(* IEC 61131-3 sources: std_i2980_v2.06_cp053/Source/IMM/ieccontrol/NozzleGeneral (part 5) *)

@F

@Trans @RT(7)Trans56 @F @T @F @F @T @F @TL(2)
TRUE

@RT(7)Trans56 @F
@Goto @RT(7)S_Ready @F @F

@Step @RT(6)Step45 @F @F @F @F @RT(0) @F
@AcbCont @RT(7)unnamed @F 0

@AltBranch @RT(3)alt @F 2
@TransSeq @RT(4)tseq @F 1
@Trans @RT(13)TNozzleNotFwd @F @T @F @F @T @F @TL(2)
NOT sv_bNozzleFwd

@RT(13)TNozzleNotFwd @F

@TransSeq @RT(4)tseq @F 4
@Trans @RT(12)TNozzleIsFwd @F @T @F @F @T @F @TL(2)
sv_bNozzleFwd

@RT(12)TNozzleIsFwd @F
@Step @RT(6)Step47 @F @F @F @F @RT(0) @F
@AcbCont @RT(7)unnamed @F 1
@Acb @RT(23)ASetContactPressBuildUp @F @T @RT(1)P @RT(0) @F @F @T @TL(2)
bContactPressBuildUp := TRUE;

@F

@Trans @RT(7)Trans71 @F @T @F @F @T @F @TL(2)
TRUE

@RT(7)Trans71 @F
@Goto @RT(24)S_CheckIfPressureBuildUp @F @F

@Step @RT(13)S_ProfileMove @F @F @F @F @RT(0) @F
@AcbCont @RT(7)unnamed @F 5
@Acb @RT(18)AResetProfileBlock @F @F @RT(1)P @RT(0) @F @F @F @F
@Acb @RT(15)AResetDetection @F @F @RT(1)P @RT(0) @F @F @F @F
@Acb @RT(11)aRunProfile @F @F @RT(1)N @RT(0) @F @F @F @F
@Acb @RT(18)ACheckContactPoint @F @F @RT(1)N @RT(0) @F @F @F @F
@Acb @RT(18)ACheckPointReached @F @F @RT(2)P0 @RT(0) @F @F @F @F

@Trans @RT(17)TProfileMoveReady @F @T @F @F @T @F @TL(2)
NOT abNozzleFwdProfile.aRun.bActive

@RT(17)TProfileMoveReady @F
@Step @RT(7)S_Check @F @F @F @F @RT(0) @F
@AcbCont @RT(7)unnamed @F 0

@AltBranch @RT(3)alt @F 2
@TransSeq @RT(4)tseq @F 1
@Trans @RT(15)TContactPointOk @F @T @F @F @T @F @TL(2)
bContactPointDetected

@RT(15)TContactPointOk @F

@TransSeq @RT(4)tseq @F 2
@Trans @RT(18)TContactPointNotOk @F @T @F @F @T @F @TL(2)
NOT bContactPointDetected

@RT(18)TContactPointNotOk @F
@Goto @RT(7)S_Ready @F @F

@Step @RT(14)S_NewPosOffset @F @F @F @F @RT(0) @F
@AcbCont @RT(7)unnamed @F 1
@Acb @RT(21)AActivateContactForce @F @T @RT(1)P @RT(0) @F @F @T @TL(2)
bContactPressBuildUp := TRUE;

@F

@Trans @RT(7)Trans45 @F @T @F @F @T @F @TL(2)
TRUE

@RT(7)Trans45 @F

@TransSeq @RT(4)tseq @F 11
@Trans @RT(12)TLimitSwitch @F @T @F @F @T @F @TL(2)
sv_MovementMode = nLimitSwitchDependent

@RT(12)TLimitSwitch @F
@Step @RT(18)S_CheckLimitSwitch @F @F @F @F @RT(0) @F
@AcbCont @RT(7)unnamed @F 1
@Acb @RT(8)Action21 @F @T @RT(1)N @RT(0) @F @F @T @TL(3)
dActiveTime := T#0s;
sv_NozzleFwdTimesAct.dActMoveTime := T#0s;

@F

@AltBranch @RT(3)alt @F 2
@TransSeq @RT(4)tseq @F 1
@Trans @RT(21)TLimitSwitchAvailable @F @T @F @F @T @F @TL(3)
mbLimitSwFwdLinked AND
NOT di_LimitSwitchFwd

@RT(21)TLimitSwitchAvailable @F

@TransSeq @RT(4)tseq @F 4
@Trans @RT(17)TStartSecondStage @F @T @F @F @T @F @TL(4)
mbLimitSwFwdLinked AND
di_LimitSwitchFwd

@RT(17)TStartSecondStage @F
@Step @RT(11)CheckLimits @F @F @F @F @RT(0) @F
@AcbCont @RT(7)unnamed @F 0

@AltBranch @RT(3)alt @F 3
@TransSeq @RT(4)tseq @F 1
@Trans @RT(12)TGoToTimeDep @F @T @F @F @T @F @TL(3)
NOT mbLimitSwFwd2Linked

@RT(12)TGoToTimeDep @F

@TransSeq @RT(4)tseq @F 2
@Trans @RT(18)TGoToSecLimitSwDep @F @T @F @F @T @F @TL(3)
mbLimitSwFwd2Linked AND
NOT di_LimitSwitchFwd2

@RT(18)TGoToSecLimitSwDep @F
@Goto @RT(16)S_ConstStage2Di2 @F @F

@TransSeq @RT(4)tseq @F 2
@Trans @RT(14)TNozzleInFront @F @T @F @F @T @F @TL(3)
mbLimitSwFwd2Linked
AND di_LimitSwitchFwd2

@RT(14)TNozzleInFront @F
@Goto @RT(29)S_ActivateContactFAfterLimSW2 @F @F

@Goto @RT(13)S_ConstStage2 @F @F

@Step @RT(13)S_ConstStage1 @F @F @F @F @RT(0) @F
@AcbCont @RT(7)unnamed @F 4
@Acb @RT(17)AResetConstStage1 @F @F @RT(1)P @RT(0) @F @F @F @F
@Acb @RT(17)ACheckVelCReached @F @F @RT(1)N @RT(0) @F @F @F @F
@Acb @RT(15)AS2PreOutputMax @F @F @RT(1)N @RT(0) @F @F @F @F
@Acb @RT(15)aRunConstStage1 @F @F @RT(1)N @RT(0) @F @F @F @F

@AltBranch @RT(3)alt @F 3
@TransSeq @RT(4)tseq @F 1
@Trans @RT(19)TLimitSwitchReached @F @T @F @F @T @F @TL(4)
di_LimitSwitchFwd AND
bVelC1Reached AND
NOT mbLimitSwFwd2Linked

@RT(19)TLimitSwitchReached @F

@TransSeq @RT(4)tseq @F 6
@Trans @RT(20)TGoToNextLimitSwitch @F @T @F @F @T @F @TL(4)
mbLimitSwFwd2Linked AND
di_LimitSwitchFwd AND
bVelC1Reached

@RT(20)TGoToNextLimitSwitch @F
@Step @RT(16)S_ConstStage2Di2 @F @F @T @F @RT(0) @F
@AcbCont @RT(7)unnamed @F 3
@Acb @RT(20)AResetConstStage2DI2 @F @F @RT(1)P @RT(0) @F @F @F @F
@Acb @RT(16)AStopConstStage1 @F @F @RT(1)N @RT(0) @F @F @F @F
@Acb @RT(18)aRunConstStage1To2 @F @F @RT(1)N @RT(0) @F @F @F @F

@Trans @RT(7)Trans44 @F @T @F @F @T @F @TL(3)
((NOT abNozzleFwdConstStage2.aRun.bActive)
AND(NOT abNozzleFwdConstStage1.aRun.bActive))

@RT(7)Trans44 @F
@Step @RT(29)S_ActivateContactFAfterLimSW2 @F @F @T @F @RT(0) @F
@AcbCont @RT(7)unnamed @F 1
@Acb @RT(24)AActivateConFAfterLimSW2 @F @T @RT(1)P @RT(0) @F @F @T @TL(4)
IF di_LimitSwitchFwd2 THEN
   bContactPressBuildUp := TRUE;
END_IF;

@F

@Trans @RT(7)Trans67 @F @T @F @F @T @F @TL(2)
TRUE

@RT(7)Trans67 @F
@Goto @RT(8)S_PreOut @F @F

@TransSeq @RT(4)tseq @F 2
@Trans @RT(7)Trans35 @F @T @F @F @T @T @TL(2)
NOT abNozzleFwdConstStage1.aRun.bActive

@RT(7)Trans35 @F
@Goto @RT(8)S_PreOut @F @F

@Step @RT(13)S_ConstStage2 @F @F @T @F @RT(0) @F
@AcbCont @RT(7)unnamed @F 3
@Acb @RT(17)AResetConstStage2 @F @F @RT(1)P @RT(0) @F @F @F @F
@Acb @RT(16)AStopConstStage1 @F @F @RT(1)N @RT(0) @F @F @F @F
@Acb @RT(15)aRunConstStage2 @F @F @RT(1)N @RT(0) @F @F @F @F

@Trans @RT(17)TConstStage2Ready @F @T @F @F @T @F @TL(3)
    (NOT abNozzleFwdConstStage2.aRun.bActive)
AND (NOT abNozzleFwdConstStage1.aRun.bActive)

@RT(17)TConstStage2Ready @F
@Step @RT(29)S_ActivateContactFAfterLimSW1 @F @F @F @F @RT(0) @F
@AcbCont @RT(7)unnamed @F 1
@Acb @RT(24)AActivateConFAfterLimSW1 @F @T @RT(1)P @RT(0) @F @F @T @TL(4)
IF (sv_dNozzleFwdStage2Act >= sv_dNozzleFwdStage2Set) THEN
   bContactPressBuildUp := TRUE;
END_IF;

@F

@Trans @RT(7)Trans68 @F @T @F @F @T @F @TL(2)
TRUE

@RT(7)Trans68 @F
@Step @RT(8)S_PreOut @F @F @T @F @RT(0) @F
@AcbCont @RT(7)unnamed @F 1
@Acb @RT(13)AS2PreOutput0 @F @F @RT(1)N @RT(0) @F @F @F @F

@Trans @RT(7)Trans21 @F @T @F @F @T @F @TL(2)
TRUE

@RT(7)Trans21 @F

@TransSeq @RT(4)tseq @F 5
@Trans @RT(9)TTimeMode @F @T @F @F @T @F @TL(2)
sv_MovementMode = nMoveTimeDependent

@RT(9)TTimeMode @F
@Step @RT(11)S_ConstTime @F @F @F @F @RT(0) @F
@AcbCont @RT(7)unnamed @F 3
@Acb @RT(6)AReset @F @F @RT(1)P @RT(0) @F @F @F @F
@Acb @RT(13)aRunConstTime @F @F @RT(1)N @RT(0) @F @F @F @F
@Acb @RT(18)ASetFwdTimeReached @F @F @RT(1)N @RT(0) @F @F @F @F

@Trans @RT(14)TTimeMoveReady @F @T @F @F @T @F @TL(2)
NOT abNozzleFwdConstStage2.aRun.bActive

@RT(14)TTimeMoveReady @F
@Step @RT(30)S_ActivateConFAfterTimeElapsed @F @F @F @F @RT(0) @F
@AcbCont @RT(7)unnamed @F 1
@Acb @RT(29)AActivateConFAfterTimeElapsed @F @T @RT(1)P @RT(0) @F @F @T @TL(2)
bContactPressBuildUp := sv_bFwdTimeReached;

@F

@Trans @RT(7)Trans64 @F @T @F @F @T @F @TL(2)
TRUE

@RT(7)Trans64 @F

@Step @RT(24)S_CheckIfPressureBuildUp @F @F @T @F @RT(0) @F
@AcbCont @RT(7)unnamed @F 0

@AltBranch @RT(3)alt @F 2
@TransSeq @RT(4)tseq @F 3
@Trans @RT(16)TMoveFwdContactF @F @T @F @F @T @F @TL(3)
g_MoveCtrl.pData^.MoveId = cMoveFwdContactF
AND bContactPressBuildUp

@RT(16)TMoveFwdContactF @F
@Step @RT(23)S_NozzlePressureBuildup @F @F @F @F @RT(0) @F
@AcbCont @RT(7)unnamed @F 2
@Acb @RT(23)AResetConstBuildUpPress @F @F @RT(1)P @RT(0) @F @F @F @F
@Acb @RT(21)aRunConstBuildUpPress @F @F @RT(1)N @RT(0) @F @F @F @F

@Trans @RT(18)TPressBuiltUpReady @F @T @F @F @T @F @TL(2)
NOT abNozzleFwdPressBuildUp.aRun.bActive

@RT(18)TPressBuiltUpReady @F

@TransSeq @RT(4)tseq @F 3
@Trans @RT(8)TMoveFwd @F @T @F @F @T @F @TL(3)
g_MoveCtrl.pData^.MoveId = cMoveFwd
OR NOT bContactPressBuildUp

@RT(8)TMoveFwd @F
@Step @RT(15)S_AdaptDuration @F @F @F @F @RT(0) @F
@AcbCont @RT(7)unnamed @F 1
@Acb @RT(18)ADurationReference @F @F @RT(1)P @RT(0) @F @F @F @F

@Trans @RT(7)Trans72 @F @T @F @F @T @F @TL(2)
TRUE

@RT(7)Trans72 @F

@Step @RT(7)S_Ready @F @F @T @F @RT(0) @F
@AcbCont @RT(7)unnamed @F 1
@Acb @RT(6)AReady @F @T @RT(1)P @RT(0) @F @F @T @TL(5)
bReady := TRUE;
fbSetMovementState(MoveId   := g_MoveCtrl.pData^.MoveId,
                   MoveDir  := g_MoveCtrl.pData^.MoveDir,
                   State    := nInactive);

@F

@Trans @RT(6)TReady @F @T @T @T @T @T @TL(2)
TRUE

@RT(6)TReady @F

@END_SfcData
@SaActions 33
@SaText @RT(16)AResetConstBlock 1 @TL(7)
(**************************************** WARNING ********************************************
 *** The KEBA Kemro K2 System including software is not intended for safety control tasks! ***
 ***                       For further information see Comment tab!                        ***
 *********************************************************************************************)

abNozzleFwdConstSetup.aRun(bStart := FALSE);

@SaText @RT(18)AResetProfileBlock 1 @TL(8)
(**************************************** WARNING ********************************************
 *** The KEBA Kemro K2 System including software is not intended for safety control tasks! ***
 ***                       For further information see Comment tab!                        ***
 *********************************************************************************************)

abNozzleFwdProfile.aRun(bStart := FALSE);

@SaText @RT(17)AResetConstStage1 1 @TL(8)
(**************************************** WARNING ********************************************
 *** The KEBA Kemro K2 System including software is not intended for safety control tasks! ***
 ***                       For further information see Comment tab!                        ***
 *********************************************************************************************)

abNozzleFwdConstStage1.aRun(bStart := FALSE);
bStage1Runned := TRUE;

@SaText @RT(17)AResetConstStage2 1 @TL(10)
(**************************************** WARNING ********************************************
 *** The KEBA Kemro K2 System including software is not intended for safety control tasks! ***
 ***                       For further information see Comment tab!                        ***
 *********************************************************************************************)
dActiveTime := sv_NozzleFwdTimesAct.dActMoveTime;
abNozzleFwdConstStage2.aRun(bStart := FALSE);

//set move time
abNozzleFwdConstStage2.aSetMoveTime(dSetMoveTime := sv_dNozzleFwdStage2Set);

@SaText @RT(16)AResetCalibBlock 1 @TL(14)
(**************************************** WARNING ********************************************
 *** The KEBA Kemro K2 System including software is not intended for safety control tasks! ***
 ***                       For further information see Comment tab!                        ***
 *********************************************************************************************)

bError := FALSE;
abNozzleFwdCalib.aRun(bStart := FALSE,
                      LintabPoint := sv_TmpLintabPoint);
IF abNozzleFwdCalib.aRun.bError THEN
   sv_CalibState.Status := tnCalibState_Error;
   bError := TRUE;
   dummy := Print("Calib Error: Reset calib block failed");
END_IF;

@SaText @RT(17)ACheckVelCReached 1 @TL(2)
bVelC1Reached := (ABS(sv_rVelocityAbs - sv_ConstFwdStage1.Velocity.Output.rOutputValue) < 0.1);

@SaText @RT(13)AS2PreOutput0 1 @TL(5)
bStage1Runned := FALSE;

sv_ConstFwdStage2.Pressure.PreOutput.rOutputValue := 0.0;
sv_ConstFwdStage2.Velocity.PreOutput.rOutputValue := 0.0;

@SaText @RT(15)AS2PreOutputMax 1 @TL(7)

IF bVelC1Reached THEN
  sv_ConstFwdStage2.Pressure.PreOutput.rOutputValue := sv_ConstFwdStage1.Pressure.Output.rOutputValue;
  sv_ConstFwdStage2.Velocity.PreOutput.rOutputValue := sv_ConstFwdStage1.Velocity.Output.rOutputValue;
END_IF;

@SaText @RT(16)AStopConstStage1 1 @TL(7)
(**************************************** WARNING ********************************************
 *** The KEBA Kemro K2 System including software is not intended for safety control tasks! ***
 ***                       For further information see Comment tab!                        ***
 *********************************************************************************************)

abNozzleFwdConstStage1.aRun(bStop:=TRUE);

@SaText @RT(16)ACheckCalibError 1 @TL(5)
IF bError THEN
   sv_CalibState.Status := tnCalibState_Error;
   dummy := Print("Calib Error: %i", iErrorInfo);
END_IF;

@SaText @RT(17)AResetAdjustBlock 1 @TL(14)
(**************************************** WARNING ********************************************
 *** The KEBA Kemro K2 System including software is not intended for safety control tasks! ***
 ***                       For further information see Comment tab!                        ***
 *********************************************************************************************)

//init supervision time
fbTSupervisionTime(IN := FALSE,
                   PT := sv_dMaxNozzleAdjustTime);

abNozzleFwdConstAdjust.aRun(bStart := FALSE);
bAutoAdjustAllowed := TRUE;

sv_rNozzlePositionOffset := 0.0;

@SaText @RT(16)AResetStandStill 1 @TL(6)
bStandStill := FALSE;

IF NOT mbLimitSwFwdLinked THEN
   fbStandStill(bDoCalib := FALSE);
END_IF;

@SaText @RT(17)ADetectStandStill 1 @TL(22)
(**************************************** WARNING ********************************************
 *** The KEBA Kemro K2 System including software is not intended for safety control tasks! ***
 ***                       For further information see Comment tab!                        ***
 *********************************************************************************************)

IF NOT bStandStill THEN
   IF mbLimitSwFwdLinked THEN
      bStandStill := di_LimitSwitchFwd;
   ELSE
      fbStandStill(rActVoltage := ai_Position,
                   bDoCalib := TRUE,
                   dCalibTime := sv_dSetStandstillDetectionTime,
                   rMaxVoltageDiff := sv_rMaxVoltageDiff,
                   bStandStill => bStandStill);
   END_IF;
END_IF;

@SaText @RT(16)ASetNozzleOffset 1 @TL(21)
(**************************************** WARNING ********************************************
 *** The KEBA Kemro K2 System including software is not intended for safety control tasks! ***
 ***                       For further information see Comment tab!                        ***
 *********************************************************************************************)

//calculate offset
//attention: offset is normally negative
sv_rNozzlePositionOffset := sv_rNozzlePositionOffset - sv_rNozzlePosition;

sv_rNozzleStrokePlaus := sv_rNozzleStroke + sv_rNozzlePositionOffset;

// automatically correct bwd profile if necessary
FOR i:=1 TO sv_NozzleBwdProfVis.Profile.iNoOfPoints + 1 DO
   sv_NozzleBwdProfVis.Profile.Points[i].rStartPos :=
         MIN(sv_NozzleBwdProfVis.Profile.Points[i].rStartPos, sv_rNozzleStrokePlaus);
END_FOR;

sv_bContactPointDetected := TRUE;
sv_bNozzleAdjHMI := FALSE;
SET_ALARM(erNozzleAdjustFinished);

@SaText @RT(23)AResetConstBuildUpPress 1 @TL(12)
(**************************************** WARNING ********************************************
*** The KEBA Kemro K2 System including software is not intended for safety control tasks! ***
***                       For further information see Comment tab!                        ***
*********************************************************************************************)

abNozzleFwdPressBuildUp.aRun(bStart := FALSE);

//set move time
abNozzleFwdPressBuildUp.aSetMoveTime(dSetMoveTime := sv_dNozzleFwdContactFSet);

sv_NozzleFwdContactFData.pdHoldDuration := @sv_dNozzleFwdContactFSet;

@SaText @RT(15)AResetDetection 1 @TL(11)
(**************************************** WARNING ********************************************
 *** The KEBA Kemro K2 System including software is not intended for safety control tasks! ***
 ***                       For further information see Comment tab!                        ***
 *********************************************************************************************)

bStandStill := FALSE;
fbStandStill(bDoCalib := FALSE);
fbRTrigStandstill(CLK := FALSE);
bContactPointDetected := FALSE;
bContactPointDetError := FALSE;

@SaText @RT(18)ACheckPointReached 1 @TL(18)
(**************************************** WARNING ********************************************
 *** The KEBA Kemro K2 System including software is not intended for safety control tasks! ***
 ***                       For further information see Comment tab!                        ***
 *********************************************************************************************)

IF abNozzleFwdProfile.aRun.bTimeOut OR abNozzleFwdProfile.aRun.bError THEN
   //timeout or error during profile movement
   bContactPointDetected := FALSE;
ELSIF (((sv_rNozzlePosition > sv_rPosOffsetTolerance) AND bStandStill)
   OR (sv_rNozzlePosition <= -sv_rPosOffsetTolerance)) THEN
   //standstill out of tolerance or movement finished out of tolerance
   bContactPointDetected := FALSE;
   SET_ALARM(erContactPointOutOfTolerance);
ELSE
   //movement finished inside the tolerance
   bContactPointDetected := TRUE;
END_IF;

@SaText @RT(18)ACheckContactPoint 1 @TL(11)
(**************************************** WARNING ********************************************
 *** The KEBA Kemro K2 System including software is not intended for safety control tasks! ***
 ***                       For further information see Comment tab!                        ***
 *********************************************************************************************)

fbStandStill(rActVoltage := ai_Position,
             bDoCalib := TRUE,
             dCalibTime := t#500ms,
             rMaxVoltageDiff := sv_rMaxVoltageDiff,
             bStandStill => bStandStill);

@SaText @RT(18)ADurationReference 1 @TL(7)
(**************************************** WARNING ********************************************
*** The KEBA Kemro K2 System including software is not intended for safety control tasks! ***
***                       For further information see Comment tab!                        ***
*********************************************************************************************)

sv_NozzleFwdContactFData.pdHoldDuration := EMPTY;

@SaText @RT(6)AReset 1 @TL(10)
(**************************************** WARNING ********************************************
 *** The KEBA Kemro K2 System including software is not intended for safety control tasks! ***
 ***                       For further information see Comment tab!                        ***
 *********************************************************************************************)

abNozzleFwdConstStage2.aRun(bStart := FALSE);

//set move time
abNozzleFwdConstStage2.aSetMoveTime(dSetMoveTime := sv_dNozzleFwdStage2Set);

@SaText @RT(18)ASetFwdTimeReached 1 @TL(7)
(**************************************** WARNING ********************************************
 *** The KEBA Kemro K2 System including software is not intended for safety control tasks! ***
 ***                       For further information see Comment tab!                        ***
 *********************************************************************************************)

sv_bFwdTimeReached := (sv_dNozzleFwdStage2Act >= sv_dNozzleFwdStage2Set)

@SaText @RT(20)AResetConstStage2DI2 1 @TL(8)
(**************************************** WARNING ********************************************
 *** The KEBA Kemro K2 System including software is not intended for safety control tasks! ***
 ***                       For further information see Comment tab!                        ***
 *********************************************************************************************)

dActiveTime := sv_NozzleFwdTimesAct.dActMoveTime;
abNozzleFwdConstStage2.aRun(bStart := FALSE);

@SaText @RT(16)AResetIdentBlock 1 @TL(3)
abNozzleFwdStep.aRun(bStart := FALSE);

@SaText @RT(16)ATransducerCalib 1 @TL(28)
(**************************************** WARNING ********************************************
 *** The KEBA Kemro K2 System including software is not intended for safety control tasks! ***
 ***                       For further information see Comment tab!                        ***
 *********************************************************************************************)

abNozzleFwdCalib.aRun(bStop := bStop OR sv_bTransducerError,
                      bStart := TRUE,
                      rActVoltage := ai_Position,
                      rMaxVoltageDiff := sv_rMaxVoltageDiff,
                      dStandStillDetectTime := sv_dStandStillDetectTime,
                      LintabPoint := sv_TmpLintabPoint,
                      rSetValue := 0.0,
                      dDelayTimeOn := sv_NozzleFwdTimesSet.dSetDelayTimePump,
                      dDelayTimeOff := sv_NozzleFwdTimesSet.dSetDelayTimeValve,
                      bActive => sv_bOutputActive,
                      rOutputPre => sv_rPressureAbs,
                      rOutputVel => sv_rVelocityAbs,
                      bPreOutputReached => sv_bPreOutputReady,
                      iErrorInfo => iErrorInfo);
sv_bDoTransducerCalib := NOT (abNozzleFwdCalib.aRun.bPointDetected);
bError := abNozzleFwdCalib.aRun.bError OR bError;

abLintabApplyPres.aCalc(rX := sv_rPressureAbs,
                        rY => sv_rPressure);

abLintabApplyVel.aCalc(rX := sv_rVelocityAbs,
                       rY => sv_rVelocity);

@SaText @RT(11)AStepOutput 1 @TL(30)
(**************************************** WARNING ********************************************
 *** The KEBA Kemro K2 System including software is not intended for safety control tasks! ***
 ***                       For further information see Comment tab!                        ***
 *********************************************************************************************)

abNozzleFwdStep.aRun(bUsePosDetect := sv_rIdentPosition <> 0.0,
                     rPositionDown := (sv_rNozzlePosition + sv_rIdentPosition) * 0.5,
                     rLowOutput := sv_rMaxSpeedFwd * 0.1,
                     bStart := TRUE,
                     bStop := bStop,
                     bDirection := FALSE,
                     rActPos := sv_rNozzlePosition,
                     rTargetPos := sv_rIdentPosition,
                     dDelayTimeOn := sv_NozzleFwdTimesSet.dSetDelayTimePump,
                     dDelayTimeOff := sv_dSetDelayTimeOffFwd,
                     rPositionUp := sv_rNozzlePosition,
                     rHighOutput := sv_ConstFwdSetup.Velocity.Output.rOutputValue,
                     dMaxMoveTime := sv_NozzleFwdTimesSet.dMaxMoveTime,
                     rStopRamp := sv_rIdentStopRamp,
                     bActive => sv_bOutputActive,
                     rOutputPre => sv_rPressureAbs,
                     rOutputVel => sv_rVelocityAbs,
                     bPreOutputReached => sv_bPreOutputReady);

abLintabApplyPres.aCalc(rX := sv_rPressureAbs,
                        rY => sv_rPressure);

abLintabApplyVel.aCalc(rX := sv_rVelocityAbs,
                       rY => sv_rVelocity);

@SaText @RT(11)aRunProfile 1 @TL(28)
(**************************************** WARNING ********************************************
 *** The KEBA Kemro K2 System including software is not intended for safety control tasks! ***
 ***                       For further information see Comment tab!                        ***
 *********************************************************************************************)

abNozzleFwdProfile.aRun(bStop := bStop OR sv_bTransducerError OR bStandStill,
                        bStart := TRUE,
                        rActPosition := sv_rNozzlePosition,
                        dMaxMoveTime := sv_NozzleFwdTimesSet.dMaxMoveTime,
                        dDelayTimeOn := sv_NozzleFwdTimesSet.dSetDelayTimePump,
                        dDelayTimeOff := sv_NozzleFwdTimesSet.dSetDelayTimeValve,
                        DeadTime := sv_dSetDelayTimeOffFwd,
                        rSmoothFactor := sv_rSmoothFactor,
                        bActive => sv_bOutputActive,
                        iActiveStage => sv_iActiveStage,
                        bPreOutputReached => sv_bPreOutputReady);

b := WRITE_SVREAL_DIRECT(sv_rPressureAbs, abNozzleFwdProfile.aRun.rPressureOutput);
b := WRITE_SVREAL_DIRECT(sv_rVelocityAbs, abNozzleFwdProfile.aRun.rVelocityOutput);
b := WRITE_SV_DIRECT(sv_NozzleFwdTimesAct.dActMoveTime, abNozzleFwdProfile.aRun.dActMoveTime);

abLintabApplyPres.aCalc(rX := sv_rPressureAbs);
b := WRITE_SVREAL_DIRECT(sv_rPressure, abLintabApplyPres.aCalc.rY);

abLintabApplyVel.aCalc(rX := sv_rVelocityAbs);
b := WRITE_SVREAL_DIRECT(sv_rVelocity, abLintabApplyVel.aCalc.rY);

@SaText @RT(13)aRunConstTime 1 @TL(26)
(**************************************** WARNING ********************************************
 *** The KEBA Kemro K2 System including software is not intended for safety control tasks! ***
 ***                       For further information see Comment tab!                        ***
 *********************************************************************************************)

abNozzleFwdConstStage2.aRun(bStart := TRUE,
                            bStop := bStop,
                            bUsePosDetect := FALSE,
                            dMaxTime := sv_NozzleFwdTimesSet.dMaxMoveTime,
                            dDelayTimeOn := sv_NozzleFwdTimesSet.dSetDelayTimePump,
                            dDelayTimeOff := sv_NozzleFwdTimesSet.dSetDelayTimeValve,
                            bActive => sv_bOutputActive,
                            bPreOutputReached => sv_bPreOutputReady);

b := WRITE_SVREAL_DIRECT(sv_rPressureAbs, abNozzleFwdConstStage2.aRun.rOutputPre);
b := WRITE_SVREAL_DIRECT(sv_rVelocityAbs, abNozzleFwdConstStage2.aRun.rOutputVel);
b := WRITE_SV_DIRECT(sv_NozzleFwdTimesAct.dActMoveTime, abNozzleFwdConstStage2.aRun.dActTime);
b := WRITE_SV_DIRECT(sv_dNozzleFwdStage2Act, sv_NozzleFwdTimesAct.dActMoveTime);

abLintabApplyPres.aCalc(rX := sv_rPressureAbs);
b := WRITE_SVREAL_DIRECT(sv_rPressure, abLintabApplyPres.aCalc.rY);

abLintabApplyVel.aCalc(rX := sv_rVelocityAbs);
b := WRITE_SVREAL_DIRECT(sv_rVelocity, abLintabApplyVel.aCalc.rY);

@SaText @RT(15)aRunConstStage2 1 @TL(43)
(**************************************** WARNING ********************************************
 *** The KEBA Kemro K2 System including software is not intended for safety control tasks! ***
 ***                       For further information see Comment tab!                        ***
 *********************************************************************************************)

IF (bStage1Runned) THEN
   dDelayTimeOn := T#0s;
   dDelayTimeOff := T#0s;
ELSE
   dDelayTimeOn := sv_NozzleFwdTimesSet.dSetDelayTimePump;
   dDelayTimeOff := sv_NozzleFwdTimesSet.dSetDelayTimeValve;
END_IF;

abNozzleFwdConstStage2.aRun(dMaxTime := sv_NozzleFwdTimesSet.dMaxMoveTime - dActiveTime,
                            bStart := TRUE,
                            bStop := bStop,
                            bUsePosDetect := FALSE,
                            dDelayTimeOn := dDelayTimeOn,
                            dDelayTimeOff := dDelayTimeOff,
                            rOutputPre => tmpPressureAbs,
                            rOutputVel => tmpVelocityAbs,
                            bActive => sv_bOutputActive,
                            bPreOutputReached => sv_bPreOutputReady);
dActMoveTime := abNozzleFwdConstStage2.aRun.dActTime + dActiveTime;
b := WRITE_SV_DIRECT(sv_NozzleFwdTimesAct.dActMoveTime, dActMoveTime);
b := WRITE_SV_DIRECT(sv_dNozzleFwdStage2Act, abNozzleFwdConstStage2.aRun.dActTime);

// sv_bPreOutput must be true for 2nd cycle, then outputvalue is valid
IF (sv_bPreOutputReady AND bPreOutputOld) THEN
   b := WRITE_SVREAL_DIRECT(sv_rPressureAbs, tmpPressureAbs);
   b := WRITE_SVREAL_DIRECT(sv_rVelocityAbs, tmpVelocityAbs);
END_IF;

bPreOutputOld := sv_bPreOutputReady;

abLintabApplyPres.aCalc(rX := sv_rPressureAbs);
b := WRITE_SVREAL_DIRECT(sv_rPressure, abLintabApplyPres.aCalc.rY);

abLintabApplyVel.aCalc(rX := sv_rVelocityAbs);
b := WRITE_SVREAL_DIRECT(sv_rVelocity, abLintabApplyVel.aCalc.rY);

@SaText @RT(18)aRunConstStage1To2 1 @TL(42)
(**************************************** WARNING ********************************************
 *** The KEBA Kemro K2 System including software is not intended for safety control tasks! ***
 ***                       For further information see Comment tab!                        ***
 *********************************************************************************************)

IF (bStage1Runned) THEN
   dDelayTimeOn := T#0s;
   dDelayTimeOff := T#0s;
ELSE
   dDelayTimeOn := sv_NozzleFwdTimesSet.dSetDelayTimePump;
   dDelayTimeOff := sv_NozzleFwdTimesSet.dSetDelayTimeValve;
END_IF;

abNozzleFwdConstStage2.aRun(bStop := bStop OR di_LimitSwitchFwd2,
                            dMaxTime := (sv_NozzleFwdTimesSet.dMaxMoveTime - dActiveTime),
                            bStart := TRUE,
                            bUsePosDetect := FALSE,
                            dDelayTimeOn := dDelayTimeOn,
                            dDelayTimeOff := dDelayTimeOff,
                            rOutputPre => tmpPressureAbs,
                            rOutputVel => tmpVelocityAbs,
                            bActive => sv_bOutputActive,
                            bPreOutputReached => sv_bPreOutputReady);
dActMoveTime := abNozzleFwdConstStage2.aRun.dActTime + dActiveTime;
b := WRITE_SV_DIRECT(sv_NozzleFwdTimesAct.dActMoveTime, dActMoveTime);

// sv_bPreOutput must be true for 2nd cycle, then outputvalue is valid
IF (sv_bPreOutputReady AND bPreOutputOld) THEN
   b := WRITE_SVREAL_DIRECT(sv_rPressureAbs, tmpPressureAbs);
   b := WRITE_SVREAL_DIRECT(sv_rVelocityAbs, tmpVelocityAbs);
END_IF;

bPreOutputOld := sv_bPreOutputReady;

abLintabApplyPres.aCalc(rX := sv_rPressureAbs);
b := WRITE_SVREAL_DIRECT(sv_rPressure, abLintabApplyPres.aCalc.rY);

abLintabApplyVel.aCalc(rX := sv_rVelocityAbs);
b := WRITE_SVREAL_DIRECT(sv_rVelocity, abLintabApplyVel.aCalc.rY);

@SaText @RT(15)aRunConstStage1 1 @TL(32)
(**************************************** WARNING ********************************************
 *** The KEBA Kemro K2 System including software is not intended for safety control tasks! ***
 ***                       For further information see Comment tab!                        ***
 *********************************************************************************************)

abNozzleFwdConstStage1.aRun(bStop := bStop OR (di_LimitSwitchFwd AND NOT bVelC1Reached),
                            bStart := TRUE,
                            bUsePosDetect := FALSE,
                            dMaxTime := sv_NozzleFwdTimesSet.dMaxMoveTime,
                            dDelayTimeOn := sv_NozzleFwdTimesSet.dSetDelayTimePump,
                            dDelayTimeOff := sv_NozzleFwdTimesSet.dSetDelayTimeValve,
                            rOutputPre => tmpPressureAbs,
                            rOutputVel => tmpVelocityAbs,
                            bActive => sv_bOutputActive,
                            bPreOutputReached => sv_bPreOutputReady);

b := WRITE_SV_DIRECT(sv_NozzleFwdTimesAct.dActMoveTime, abNozzleFwdConstStage1.aRun.dActTime);

// sv_bPreOutput must be true for 2nd cycle, then outputvalue is valid
IF (sv_bPreOutputReady AND bPreOutputOld) THEN
   b := WRITE_SVREAL_DIRECT(sv_rPressureAbs, tmpPressureAbs);
   b := WRITE_SVREAL_DIRECT(sv_rVelocityAbs, tmpVelocityAbs);
END_IF;

bPreOutputOld := sv_bPreOutputReady;

abLintabApplyPres.aCalc(rX := sv_rPressureAbs);
b := WRITE_SVREAL_DIRECT(sv_rPressure, abLintabApplyPres.aCalc.rY);

abLintabApplyVel.aCalc(rX := sv_rVelocityAbs);
b := WRITE_SVREAL_DIRECT(sv_rVelocity, abLintabApplyVel.aCalc.rY);

@SaText @RT(14)aRunConstSetup 1 @TL(22)
(**************************************** WARNING ********************************************
 *** The KEBA Kemro K2 System including software is not intended for safety control tasks! ***
 ***                       For further information see Comment tab!                        ***
 *********************************************************************************************)

abNozzleFwdConstSetup.aRun(bStart := TRUE,
                           bStop := bStop,
                           bUsePosDetect := FALSE,
                           dDelayTimeOn := sv_NozzleFwdTimesSet.dSetDelayTimePump,
                           dDelayTimeOff := sv_NozzleFwdTimesSet.dSetDelayTimeValve,
                           rOutputPre => sv_rPressureAbs,
                           rOutputVel => sv_rVelocityAbs,
                           bActive => sv_bOutputActive,
                           dActTime => sv_NozzleFwdTimesAct.dActMoveTime,
                           bPreOutputReached => sv_bPreOutputReady);

abLintabApplyPres.aCalc(rX := sv_rPressureAbs,
                        rY => sv_rPressure);

abLintabApplyVel.aCalc(rX := sv_rVelocityAbs,
                       rY => sv_rVelocity);

@SaText @RT(21)aRunConstBuildUpPress 1 @TL(27)
(**************************************** WARNING ********************************************
 *** The KEBA Kemro K2 System including software is not intended for safety control tasks! ***
 ***                       For further information see Comment tab!                        ***
 *********************************************************************************************)

abNozzleFwdPressBuildUp.aRun(bStart := TRUE,
                             bStop := bStop,
                             bUsePosDetect := FALSE,
                             dMaxTime := sv_NozzleFwdTimesSet.dMaxMoveTime,
                             dDelayTimeOn := sv_NozzleFwdTimesSet.dSetDelayTimePump,
                             dDelayTimeOff := sv_NozzleFwdTimesSet.dSetDelayTimeValve,
                             bActive => sv_bOutputActive,
                             bPreOutputReached => sv_bPreOutputReady);

sv_bPressBuildUpActive := sv_bOutputActive;
b := WRITE_SVREAL_DIRECT(sv_rPressureAbs, abNozzleFwdPressBuildUp.aRun.rOutputPre);
b := WRITE_SVREAL_DIRECT(sv_rVelocityAbs, abNozzleFwdPressBuildUp.aRun.rOutputVel);
b := WRITE_SV_DIRECT(sv_dActPressureBuildUpTime, abNozzleFwdPressBuildUp.aRun.dActTime);
b := WRITE_SV_DIRECT(sv_dNozzleFwdContactFAct, sv_dActPressureBuildUpTime);

abLintabApplyPres.aCalc(rX := sv_rPressureAbs);
b := WRITE_SVREAL_DIRECT(sv_rPressure, abLintabApplyPres.aCalc.rY);

abLintabApplyVel.aCalc(rX := sv_rVelocityAbs);
b := WRITE_SVREAL_DIRECT(sv_rVelocity, abLintabApplyVel.aCalc.rY);

@SaText @RT(20)aRunConstAdjustSetup 1 @TL(25)
(**************************************** WARNING ********************************************
 *** The KEBA Kemro K2 System including software is not intended for safety control tasks! ***
 ***                       For further information see Comment tab!                        ***
 *********************************************************************************************)

abNozzleFwdConstAdjust.aRun(bStop := bStop OR bStandStill OR sv_bTransducerError OR NOT bAutoAdjustAllowed,
                            bStart := TRUE,
                            bUsePosDetect := FALSE,
                            dMaxTime := sv_NozzleFwdTimesSet.dMaxMoveTime,
                            dDelayTimeOn := sv_NozzleFwdTimesSet.dSetDelayTimePump,
                            dDelayTimeOff := sv_NozzleFwdTimesSet.dSetDelayTimeValve,
                            rOutputPre => sv_rPressureAbs,
                            rOutputVel => sv_rVelocityAbs,
                            bActive => sv_bOutputActive,
                            dActTime => sv_NozzleFwdTimesAct.dActMoveTime,
                            bPreOutputReached => sv_bPreOutputReady);

abLintabApplyPres.aCalc(rX := sv_rPressureAbs,
                        rY => sv_rPressure);

abLintabApplyVel.aCalc(rX := sv_rVelocityAbs,
                       rY => sv_rVelocity);

@SaTrans 0
@SaExits 0
@END_SfcBody

@@@BEG_Comment@@@
@TL(0)

@@@END_Comment@@@

@BEG_Body
@TL(8)
(**************************************** WARNING ********************************************
 *** The KEBA Kemro K2 System including software is not intended for safety control tasks! ***
 ***                       For further information see Comment tab!                        ***
 *********************************************************************************************)

//copy stroke to start position of first profile point
sv_NozzleFwdProfVis.Profile.Points[1].rStartPos := sv_rNozzleStroke;

@END_Body

@@@BEG_Comment@@@
@TL(0)

@@@END_Comment@@@

@BEG_Body
@TL(15)
fuName := GET_MY_FU_NAME();
variableName := CONCAT(fuName,'.Fwd.rSetPressure bar');
swoState := KSWO_AddVariable( Task := TaskAnalog,
                              Name := variableName,
                              Variable := sv_rPressureAbs);
variableName := CONCAT(fuName,'.Fwd.rSetVelocity mm/s');
swoState := KSWO_AddVariable( Task := TaskAnalog,
                              Name := variableName,
                              Variable := sv_rVelocityAbs);
variableName := CONCAT(fuName,'.Fwd.bActive');
swoState := KSWO_AddVariable( Task := TaskAnalog,
                              Name := variableName,
                              Variable := sv_bOutputActive);
STOP_PROCESS_ALGORITHM();

@END_Body

@@@BEG_Comment@@@
@TL(0)

@@@END_Comment@@@

@BEG_Body
@TL(12)
(**************************************** WARNING ********************************************
 *** The KEBA Kemro K2 System including software is not intended for safety control tasks! ***
 ***                       For further information see Comment tab!                        ***
 *********************************************************************************************)

IF sv_MovementMode = nMoveTimeDependent THEN
   sv_NozzleFwdContactFData.pdInjectDuration := @sv_dNozzleFwdStage2Set;
ELSE
   sv_NozzleFwdContactFData.pdInjectDuration := @sv_dCalculatedDurationFwd;
END_IF;

@END_Body

@@@BEG_Comment@@@
@TL(0)

@@@END_Comment@@@

@BEG_Body
@TL(8)
(**************************************** WARNING ********************************************
 *** The KEBA Kemro K2 System including software is not intended for safety control tasks! ***
 ***                       For further information see Comment tab!                        ***
 *********************************************************************************************)

//update sv_rNozzleStrokePlaus (used for plaus on HMI)
sv_rNozzleStrokePlaus := sv_rNozzleStroke + sv_rNozzlePositionOffset;

@END_Body

@@@BEG_Comment@@@
@TL(0)

@@@END_Comment@@@

@BEG_Body
@TL(5)
FOR i:= 3 TO 20 DO
    sv_NozzleFwdProfVis.Profile.Points[i].rVelRamp := sv_NozzleFwdProfVis.Profile.Points[2].rVelRamp;
END_FOR;

@END_Body

@@@BEG_Comment@@@
@TL(0)

@@@END_Comment@@@

@BEG_Body
@TL(21)
(**************************************** WARNING ********************************************
 *** The KEBA Kemro K2 System including software is not intended for safety control tasks! ***
 ***                       For further information see Comment tab!                        ***
 *********************************************************************************************)

//deactive movement NozzleFwdContactF in HA and FA mode
//if nozzle is already forward and contact force build up time is 0.0 sec
IF (sv_OperationMode = nSetup) OR (sv_OperationMode = nManual) OR (sv_dNozzleFwdContactFSet > t#0.0s) THEN
   sv_MoveFwdContactF.pbActivated := @sv_bTRUE;
ELSE
   //HA or FA active and set set for contact forec build up = 0 sec.
   IF ((sv_MovementMode = nMoveTimeDependent) AND sv_bFwdTimeReached) OR
      ((sv_MovementMode <> nMoveTimeDependent) AND sv_bNozzleFwd) THEN
      // nozzle is already forward -> deactivate
      sv_MoveFwdContactF.pbActivated := @sv_bFALSE;
   ELSE
      // nozzle not forward -> activate
      sv_MoveFwdContactF.pbActivated := @sv_bTRUE;
   END_IF;
END_IF;

@END_Body

@@@BEG_Comment@@@
@TL(0)

@@@END_Comment@@@
@END_Body

@END_Contents

(* ---- ABMovementAdmin.pu ---- *)
IMPORT_OVER_LISTFILE
 STOP_PROCESS_ALGORITHM
, WRITE_SV_DIRECT
, cMoveFwd
, cMoveBwd
, cCompShutOffNozzle
, cSubOpNozzleTransducer
, cMoveFwdContactF
, ABMoveBwd
, ABMoveFwd
, tsMoveCtrl
, ABOutputRequest
, tOptionId
, tnOperationMode
, tsCalibMovement
, tsRequiredPumps
, tsHydrMaxValues
, KAPPL_LintabData
, tsCylinderData
, ABCalcHydrMaxValues
, ABUpdateRelLintabPre
, ABUpdateRelLintabVel

END_IMPORT

ALGORITHM_BLOCK ABMovementAdmin #DUMMY_EDIT_BLOCK

SYSTEM_VAR
 sv_bInitStart : BOOL;
 sv_bDeviceStart : BOOL (* Start Device *);
 ai_Position : REAL;
 sv_Options : tOptionId;
 sv_bTransducerAvailable : BOOL;
 sv_iActiveStage : DINT;
 sv_iActiveStageFwd : DINT (* active profile stage mold close (fwd) *);
 sv_iActiveStageBwd : DINT (* active profile stage mold open (bwd) *);
 sv_bDeviceReady : BOOL;
 sv_OperationMode : tnOperationMode;
 sv_CalibState : tsCalibMovement;
 sv_dActFwdTime : TIME (* actual nozzle fwd time (includes contact force build up) *);
 sv_RequiredPumpsFwd : tsRequiredPumps;
 sv_RequiredPumpsBwd : tsRequiredPumps;
 sv_HydrMaxValuesFwd : tsHydrMaxValues (* hydraulic max values for nozzle fwd *);
 sv_HydrMaxValuesBwd : tsHydrMaxValues (* hydraulic max values for nozzle bwd *);
 sv_bInitDone : BOOL;
 sv_LintabOutFwdP : KAPPL_LintabData;
 sv_LintabOutFwdV : KAPPL_LintabData;
 sv_LintabOutBwdP : KAPPL_LintabData;
 sv_LintabOutBwdV : KAPPL_LintabData;
 sv_rMaxSpeedFwd : REAL;
 sv_rMaxSpeedBwd : REAL;
 sv_CylinderData : tsCylinderData;
 sv_rMaxPressureFwd : REAL;
 sv_rMaxPressureBwd : REAL;
 sv_rMaxSpeedFwdCalc : REAL;
 sv_rMaxSpeedBwdCalc : REAL;
 sv_rMaxSpeedFwdCalib : REAL;
 sv_rMaxSpeedBwdCalib : REAL;
 sv_rMaxSpeedReducePercent : REAL;
 sv_bFALSE : BOOL;
END_VAR

SYSTEM_OBJECT
 PU_Task_7 : TASK;
 TaskAnalog : TASK;
 EV_Task_1 : TASK;
 PU_Task_3 : TASK;
END_OBJECT

VAR_EXTERNAL
 g_MoveCtrl : tsMoveCtrl;
END_VAR

VAR
 abMoveBwd : ABMoveBwd;
 abMoveFwd : ABMoveFwd;
 abOutputRequest : ABOutputRequest;
 miDigitsToFloor : SINT := 2;
END_VAR

(*
Calls the registration-algo of every movementblock after the deviceregistration succeeded(sv_bInitStart->true)

*)

POSTUPDATE_ALGORITHM pInitStart ON PU_Task_7 WITH sv_bInitStart

VAR
 abCalcMaxValuesFwd : ABCalcHydrMaxValues;
 abCalcMaxValuesBwd : ABCalcHydrMaxValues;
END_VAR
#BEGIN_EDIT_BLOCK
(**************************************** WARNING ********************************************
 *** The KEBA Kemro K2 System including software is not intended for safety control tasks! ***
 ***                       For further information see Comment tab!                        ***
 *********************************************************************************************)

IF sv_bInitStart THEN

   //check if transducer is available
   sv_bTransducerAvailable := IS_LINKED(ai_Position);
   IF (sv_bTransducerAvailable) THEN
      sv_Options := sv_Options OR cSubOpNozzleTransducer;
      //set auto-calib transducer
      sv_CalibState.prInputSensor := @ai_Position;
   END_IF;

   //register and init nozzle bwd movement
   abMoveBwd.aRegister();
   abMoveBwd.aInit();

   //register and init nozzle fwd movement
   abMoveFwd.aRegister();
   abMoveFwd.aInit();

   //init calculation of hydraulic max values for nozzle fwd
   abCalcMaxValuesFwd.aInit(pRequiredPumps := @sv_RequiredPumpsFwd,
                            pHydrMaxValues := @sv_HydrMaxValuesFwd);

   //init calculation of hydraulic max values for nozzle bwd
   abCalcMaxValuesBwd.aInit(pRequiredPumps := @sv_RequiredPumpsBwd,
                            pHydrMaxValues := @sv_HydrMaxValuesBwd);

END_IF;

;#END_EDIT_BLOCK END_ALGORITHM

(*
Starts the algo paRun when sv_bDeviceStart is set by ABControl.
*)

POSTUPDATE_ALGORITHM pDeviceStart ON EV_Task_1 WITH sv_bDeviceStart

#BEGIN_EDIT_BLOCK
(**************************************** WARNING ********************************************
 *** The KEBA Kemro K2 System including software is not intended for safety control tasks! ***
 ***                       For further information see Comment tab!                        ***
 *********************************************************************************************)

IF sv_bDeviceStart THEN
   //start device
   START_PROCESS_ALGORITHM(paRun);
END_IF;

;#END_EDIT_BLOCK END_ALGORITHM

POSTUPDATE_ALGORITHM pInitRelLintabUpdater ON PU_Task_7 WITH sv_bInitDone

VAR
 abUpdateRelLintabPreFwd : ABUpdateRelLintabPre;
 abUpdateRelLintabVelFwd : ABUpdateRelLintabVel;
 abUpdateRelLintabPreBwd : ABUpdateRelLintabPre;
 abUpdateRelLintabVelBwd : ABUpdateRelLintabVel;
END_VAR
#BEGIN_EDIT_BLOCK
(**************************************** WARNING ********************************************
 *** The KEBA Kemro K2 System including software is not intended for safety control tasks! ***
 ***                       For further information see Comment tab!                        ***
 *********************************************************************************************)

abUpdateRelLintabPreFwd.aInit(pLintabOut := @sv_LintabOutFwdP,
                              prMaxPressure := @sv_rMaxPressureFwd,
                              prMaxHydrPressure := @sv_HydrMaxValuesFwd.rMaxPressure,
                              bUseForce := TRUE,
                              bFwd := TRUE,
                              pCylinderData := @sv_CylinderData);

abUpdateRelLintabVelFwd.aInit(pLintabOut := @sv_LintabOutFwdV,
                              prMaxSpeed := @sv_rMaxSpeedFwd,
                              prMaxSpeedCalc := @sv_rMaxSpeedFwdCalc,
                              prMaxSpeedCalib := @sv_rMaxSpeedFwdCalib,
                              prMaxSpeedReducePercent := @sv_rMaxSpeedReducePercent,
                              iMaxSpeedDigitsToFloor := miDigitsToFloor,
                              prAbsFlow := @sv_HydrMaxValuesFwd.rAbsFlow,
                              bFwd := TRUE,
                              pCylinderData := @sv_CylinderData);

abUpdateRelLintabPreBwd.aInit(pLintabOut := @sv_LintabOutBwdP,
                              prMaxPressure := @sv_rMaxPressureBwd,
                              prMaxHydrPressure := @sv_HydrMaxValuesBwd.rMaxPressure,
                              bUseForce := TRUE,
                              bFwd := FALSE,
                              pCylinderData := @sv_CylinderData);

abUpdateRelLintabVelBwd.aInit(pLintabOut := @sv_LintabOutBwdV,
                              prMaxSpeed := @sv_rMaxSpeedBwd,
                              prMaxSpeedCalc := @sv_rMaxSpeedBwdCalc,
                              prMaxSpeedCalib := @sv_rMaxSpeedBwdCalib,
                              prMaxSpeedReducePercent := @sv_rMaxSpeedReducePercent,
                              iMaxSpeedDigitsToFloor := miDigitsToFloor,
                              prAbsFlow := @sv_HydrMaxValuesBwd.rAbsFlow,
                              bFwd := FALSE,
                              pCylinderData := @sv_CylinderData);

;#END_EDIT_BLOCK END_ALGORITHM

(*
Calls depending on the MoveId and MoveDir the movementblock. g_MoveCtrl.MoveId/MoveDir are set by the Block ABControl after
evStart was received. The movement-block has to be called until the it returns abMoveXxx.aRun.bReady.
In case of hydraulic movements the output-request has to be done before starting the movement.
*)

PROCESS_ALGORITHM paRun ON TaskAnalog(5000)

VAR_TEMP
 dActFwdTime : TIME;
 b : BOOL;
END_VAR

(* IecGraph-Code *)

(* init step *)
INITIAL_STEP START:
Action18 (P);
END_STEP

ACTION Action18: #BEGIN_EDIT_BLOCK
b := WRITE_SV_DIRECT(sv_bDeviceStart, sv_bFALSE);

;#END_EDIT_BLOCK END_ACTION (*Action18*)

(* steps *)
STEP OUTPUT_REQUEST:
AOutputRequest (P);
ACheckOutput (N);
END_STEP

ACTION AOutputRequest: #BEGIN_EDIT_BLOCK
abOutputRequest.aRequest(pMoveData := g_MoveCtrl.pData,
                         AnaOutputMode := nAnaOutputModeMid);

;#END_EDIT_BLOCK END_ACTION (*AOutputRequest*)
ACTION ACheckOutput: #BEGIN_EDIT_BLOCK
abOutputRequest.aCheck();

;#END_EDIT_BLOCK END_ACTION (*ACheckOutput*)
STEP OUTPUT:
END_STEP

STEP BWD:
aBwd (N);
END_STEP

STEP FWD:
aFwd (N);
END_STEP

STEP READY:
Action2 (P);
END_STEP

ACTION Action2: #BEGIN_EDIT_BLOCK
abOutputRequest.aRelease(pMoveData := g_MoveCtrl.pData);
g_MoveCtrl.bReady := TRUE;
IF NOT sv_bDeviceStart THEN
    STOP_PROCESS_ALGORITHM();
END_IF;

;#END_EDIT_BLOCK END_ACTION (*Action2*)

(* transitions *)
GO_ON_TRANSITION TStart (* Trans12 *) FROM START TO OUTPUT_REQUEST :=  #BEGIN_EDIT_BLOCK
TRUE
;#END_EDIT_BLOCK
END_TRANSITION

TRANSITION Trans13 (* Trans13 *) FROM OUTPUT_REQUEST TO READY :=  #BEGIN_EDIT_BLOCK
g_MoveCtrl.bStop
;#END_EDIT_BLOCK
END_TRANSITION

GO_ON_TRANSITION Trans15 (* Trans15 *) FROM OUTPUT_REQUEST TO OUTPUT :=  #BEGIN_EDIT_BLOCK
abOutputRequest.aCheck.bReady
;#END_EDIT_BLOCK
END_TRANSITION

GO_ON_TRANSITION Trans9 (* Trans9 *) FROM OUTPUT TO BWD :=  #BEGIN_EDIT_BLOCK
g_MoveCtrl.pData^.MoveDir = cMoveBwd
;#END_EDIT_BLOCK
END_TRANSITION

GO_ON_TRANSITION TBwdReady (* Trans1 *) FROM BWD TO READY :=  #BEGIN_EDIT_BLOCK
abMoveBwd.aRun.bReady;
;#END_EDIT_BLOCK
END_TRANSITION

GO_ON_TRANSITION Trans2 (* Trans2 *) FROM OUTPUT TO FWD :=  #BEGIN_EDIT_BLOCK
g_MoveCtrl.pData^.MoveDir = cMoveFwd
;#END_EDIT_BLOCK
END_TRANSITION

GO_ON_TRANSITION TFwdReady (* Trans11 *) FROM FWD TO READY :=  #BEGIN_EDIT_BLOCK
abMoveFwd.aRun.bReady
;#END_EDIT_BLOCK
END_TRANSITION

TRANSITION Trans8 (* Trans8 *) FROM READY TO START :=  #BEGIN_EDIT_BLOCK
TRUE
;#END_EDIT_BLOCK
END_TRANSITION

(* end IecGraph-Code *)
(* sfc-code *)

(* stand alone actions *)
ACTION aBwd: #BEGIN_EDIT_BLOCK
(**************************************** WARNING ********************************************
 *** The KEBA Kemro K2 System including software is not intended for safety control tasks! ***
 ***                       For further information see Comment tab!                        ***
 *********************************************************************************************)

abMoveBwd.aRun(bStop := g_MoveCtrl.bStop);

;#END_EDIT_BLOCK END_ACTION (*aBwd*)
ACTION aFwd: #BEGIN_EDIT_BLOCK
abMoveFwd.aRun(bStop := g_MoveCtrl.bStop);

IF g_MoveCtrl.pData^.MoveId = cMoveFwdContactF THEN
   dActFwdTime := FWD.T;
   b := WRITE_SV_DIRECT(sv_dActFwdTime, dActFwdTime);
END_IF;

;#END_EDIT_BLOCK END_ACTION (*aFwd*)
(* end sfc-code *)

END_ALGORITHM

POSTUPDATE_ALGORITHM pActiveProfileStage ON PU_Task_3 WITH sv_iActiveStage,sv_bDeviceReady

#BEGIN_EDIT_BLOCK
(**************************************** WARNING ********************************************
 *** The KEBA Kemro K2 System including software is not intended for safety control tasks! ***
 ***                       For further information see Comment tab!                        ***
 *********************************************************************************************)

IF NOT sv_bDeviceReady THEN

   IF sv_OperationMode = nSetup THEN
      //movement in setup mode active
      //-> reset active stage information
      sv_iActiveStageFwd := 0;
      sv_iActiveStageBwd := 0;
   ELSE

      //nozzle movement in manual - half - or fullauto mode
      IF g_MoveCtrl.pData^.MoveDir = cMoveFwd THEN

         //reset bwd stage info if fwd movement is started
         sv_iActiveStageBwd := 0;

         IF sv_iActiveStage > 0 THEN
            sv_iActiveStageFwd := sv_iActiveStage;
         END_IF;

      ELSIF g_MoveCtrl.pData^.MoveDir = cMoveBwd THEN

         //reset Fwd stage info if bwd movement is started
         sv_iActiveStageFwd := 0;

         IF sv_iActiveStage > 0 THEN
            sv_iActiveStageBwd := sv_iActiveStage;
         END_IF;
      END_IF;
   END_IF;

END_IF;

;#END_EDIT_BLOCK END_ALGORITHM

END_ALGORITHM_BLOCK

#END_OF_IEC_PART

@Puma @IecEditor 6 97 @Pou 25
@@@BEG_Comment@@@

@@@END_Comment@@@

@BEG_Contents

@BEG_Func
@RT(17)FuncTreeContainer
2
@Var @RT(22)STOP_PROCESS_ALGORITHM @RT(0) @T @T @DERIVED 0 @F @RT(23)KEBA_STANDARD_PROCEDURE @F
@T
@BEG_Attrib
0 @RT(0) @RT(0)
@END_Attrib
1 1 @F @F @F @F

@Var @RT(15)WRITE_SV_DIRECT @RT(0) @T @T @DERIVED 0 @F @RT(22)KEBA_STANDARD_FUNCTION @F
@T
@BEG_Attrib
0 @RT(0) @RT(0)
@END_Attrib
1 1 @F @F @F @F

@END_Func

@BEG_Const
@RT(18)ConstTreeContainer
5
@Var @RT(8)cMoveFwd @RT(0) @T @F @DT @RT(4)DINT @RT(0) @T @T @BASIC 0 @F
@F @F
@T
@BEG_Attrib
0 @RT(2)12 @RT(16)movement forward
@END_Attrib
1 1 @F @F @F @F

@Var @RT(8)cMoveBwd @RT(0) @T @F @DT @RT(4)DINT @RT(0) @T @T @BASIC 0 @F
@F @F
@T
@BEG_Attrib
0 @RT(2)11 @RT(17)movement backward
@END_Attrib
1 1 @F @F @F @F

@Var @RT(18)cCompShutOffNozzle @RT(0) @T @F @DT @RT(4)DINT @RT(0) @T @T @BASIC 0 @F
@F @F
@T
@BEG_Attrib
0 @RT(3)138 @RT(28)Component Shutter for Nozzle
@END_Attrib
1 1 @F @F @F @F

@Var @RT(22)cSubOpNozzleTransducer @RT(0) @T @F @DT @RT(5)DWORD @RT(0) @T @T @BASIC 0 @F
@F @F
@T
@BEG_Attrib
0 @RT(6)16#100 @RT(21)Nozzle has transducer
@END_Attrib
1 1 @F @F @F @F

@Var @RT(16)cMoveFwdContactF @RT(0) @T @F @DT @RT(4)DINT @RT(0) @T @T @BASIC 0 @F
@F @F
@T
@BEG_Attrib
0 @RT(2)66 @RT(45)nozzle forward with building up contact force
@END_Attrib
1 1 @F @F @F @F

@END_Const

@BEG_Export

@BEG_Kind
@ALGORITHM_BLOCK @RT(15)ABMovementAdmin @STRUCTURED_TEXT
@RT(0) @RT(0) @RT(0)
@END_Kind

@BEG_Dcl
@RT(16)DclTreeContainer
41
@Var @RT(9)abMoveBwd @RT(0) @T @T @DERIVED 0 @T @T @DT @RT(9)ABMoveBwd @RT(0) @T @T @UNKNOWN 0 @F
@F @F
@T
@BEG_Attrib
3 @RT(0) @RT(0) @RT(0)
@END_Attrib
1 0 @F @F @F @F

@Var @RT(9)abMoveFwd @RT(0) @T @T @DERIVED 0 @T @T @DT @RT(9)ABMoveFwd @RT(0) @T @T @UNKNOWN 0 @F
@F @F
@T
@BEG_Attrib
3 @RT(0) @RT(0) @RT(0)
@END_Attrib
1 0 @F @F @F @F

@Var @RT(13)sv_bInitStart @RT(0) @T @F @DT @RT(4)BOOL @RT(0) @T @T @BASIC 0 @F
@F @F
@T
@BEG_Attrib
3 @RT(0) @RT(0) @RT(0)
@END_Attrib
1 8 @F @F @F @F

@Var @RT(15)sv_bDeviceStart @RT(0) @T @F @DT @RT(4)BOOL @RT(0) @T @T @BASIC 0 @F
@F @F
@T
@BEG_Attrib
3 @RT(0) @RT(12)Start Device @RT(0)
@END_Attrib
1 8 @F @F @F @F

@Var @RT(10)g_MoveCtrl @RT(0) @T @T @DERIVED 0 @T @T @DT @RT(10)tsMoveCtrl @RT(0) @T @T @UNKNOWN 0 @F
@F @F
@T
@BEG_Attrib
3 @RT(0) @RT(0) @RT(0)
@END_Attrib
1 6 @F @F @F @F

@Var @RT(9)PU_Task_7 @RT(0) @T @T @RENAMED 0 @T @T @DT @RT(4)TASK @RT(0) @T @T @BASIC 0 @F
@F @F
@T
@BEG_Attrib
3 @RT(0) @RT(0) @RT(0)
@END_Attrib
1 7 @F @F @F @F

@Var @RT(15)abOutputRequest @RT(0) @T @T @DERIVED 0 @T @T @DT @RT(15)ABOutputRequest @RT(0) @T @T @UNKNOWN 0 @F
@F @F
@T
@BEG_Attrib
3 @RT(0) @RT(0) @RT(0)
@END_Attrib
1 0 @F @F @F @F

@Var @RT(10)TaskAnalog @RT(0) @T @T @RENAMED 0 @T @T @DT @RT(4)TASK @RT(0) @T @T @BASIC 0 @F
@F @F
@T
@BEG_Attrib
3 @RT(0) @RT(0) @RT(0)
@END_Attrib
1 7 @F @F @F @F

@Var @RT(11)ai_Position @RT(0) @T @F @DT @RT(4)REAL @RT(0) @T @T @BASIC 0 @F
@F @F
@T
@BEG_Attrib
3 @RT(0) @RT(0) @RT(0)
@END_Attrib
1 8 @F @F @F @F

@Var @RT(10)sv_Options @RT(0) @T @T @DERIVED 0 @T @T @DT @RT(9)tOptionId @RT(0) @T @T @UNKNOWN 0 @F
@F @F
@T
@BEG_Attrib
3 @RT(0) @RT(0) @RT(0)
@END_Attrib
1 8 @F @F @F @F

@Var @RT(23)sv_bTransducerAvailable @RT(0) @T @F @DT @RT(4)BOOL @RT(0) @T @T @BASIC 0 @F
@F @F
@T
@BEG_Attrib
3 @RT(0) @RT(0) @RT(0)
@END_Attrib
1 8 @F @F @F @F

@Var @RT(9)EV_Task_1 @RT(0) @T @T @RENAMED 0 @T @T @DT @RT(4)TASK @RT(0) @T @T @BASIC 0 @F
@F @F
@T
@BEG_Attrib
3 @RT(0) @RT(0) @RT(0)
@END_Attrib
1 7 @F @F @F @F

@Var @RT(9)PU_Task_3 @RT(0) @T @F @DT @RT(4)TASK @RT(0) @T @T @BASIC 0 @F
@F @F
@T
@BEG_Attrib
3 @RT(0) @RT(0) @RT(0)
@END_Attrib
1 7 @F @F @F @F

@Var @RT(15)sv_iActiveStage @RT(0) @T @F @DT @RT(4)DINT @RT(0) @T @T @BASIC 0 @F
@F @F
@T
@BEG_Attrib
3 @RT(0) @RT(0) @RT(0)
@END_Attrib
1 8 @F @F @F @F

@Var @RT(18)sv_iActiveStageFwd @RT(0) @T @F @DT @RT(4)DINT @RT(0) @T @T @BASIC 0 @F
@F @F
@T
@BEG_Attrib
3 @RT(0) @RT(37)active profile stage mold close (fwd) @RT(0)
@END_Attrib
1 8 @F @F @F @F

@Var @RT(18)sv_iActiveStageBwd @RT(0) @T @F @DT @RT(4)DINT @RT(0) @T @T @BASIC 0 @F
@F @F
@T
@BEG_Attrib
3 @RT(0) @RT(36)active profile stage mold open (bwd) @RT(0)
@END_Attrib
1 8 @F @F @F @F

@Var @RT(15)sv_bDeviceReady @RT(0) @T @F @DT @RT(4)BOOL @RT(0) @T @T @BASIC 0 @F
@F @F
@T
@BEG_Attrib
3 @RT(0) @RT(0) @RT(0)
@END_Attrib
1 8 @F @F @F @F

@Var @RT(16)sv_OperationMode @RT(0) @T @T @DERIVED 0 @T @T @DT @RT(15)tnOperationMode @RT(0) @T @T @UNKNOWN 0 @F
@F @F
@T
@BEG_Attrib
3 @RT(0) @RT(0) @RT(0)
@END_Attrib
1 8 @F @F @F @F

@Var @RT(13)sv_CalibState @RT(0) @T @T @DERIVED 0 @T @T @DT @RT(15)tsCalibMovement @RT(0) @T @T @UNKNOWN 0 @F
@F @F
@T
@BEG_Attrib
3 @RT(0) @RT(0) @RT(0)
@END_Attrib
1 8 @F @F @F @F

@Var @RT(14)sv_dActFwdTime @RT(0) @T @F @DT @RT(4)TIME @RT(0) @T @T @BASIC 0 @F
@F @F
@T
@BEG_Attrib
3 @RT(0) @RT(56)actual nozzle fwd time (includes contact force build up) @RT(0)
@END_Attrib
1 8 @F @F @F @F

@Var @RT(19)sv_RequiredPumpsFwd @RT(0) @T @T @DERIVED 0 @T @T @DT @RT(15)tsRequiredPumps @RT(0) @T @T @UNKNOWN 0 @F
@F @F
@T
@BEG_Attrib
3 @RT(0) @RT(0) @RT(0)
@END_Attrib
1 8 @F @F @F @F

@Var @RT(19)sv_RequiredPumpsBwd @RT(0) @T @T @DERIVED 0 @T @T @DT @RT(15)tsRequiredPumps @RT(0) @T @T @UNKNOWN 0 @F
@F @F
@T
@BEG_Attrib
3 @RT(0) @RT(0) @RT(0)
@END_Attrib
1 8 @F @F @F @F

@Var @RT(19)sv_HydrMaxValuesFwd @RT(0) @T @T @DERIVED 0 @T @T @DT @RT(15)tsHydrMaxValues @RT(0) @T @T @UNKNOWN 0 @F
@F @F
@T
@BEG_Attrib
3 @RT(0) @RT(35)hydraulic max values for nozzle fwd @RT(0)
@END_Attrib
1 8 @F @F @F @F

@Var @RT(19)sv_HydrMaxValuesBwd @RT(0) @T @T @DERIVED 0 @T @T @DT @RT(15)tsHydrMaxValues @RT(0) @T @T @UNKNOWN 0 @F
@F @F
@T
@BEG_Attrib
3 @RT(0) @RT(35)hydraulic max values for nozzle bwd @RT(0)
@END_Attrib
1 8 @F @F @F @F

@Var @RT(12)sv_bInitDone @RT(0) @T @F @DT @RT(4)BOOL @RT(0) @T @T @BASIC 0 @F
@F @F
@T
@BEG_Attrib
3 @RT(0) @RT(0) @RT(0)
@END_Attrib
1 8 @F @F @F @F

@Var @RT(16)sv_LintabOutFwdP @RT(0) @T @T @DERIVED 0 @T @T @DT @RT(16)KAPPL_LintabData @RT(0) @T @T @UNKNOWN 0 @F
@F @F
@T
@BEG_Attrib
3 @RT(0) @RT(0) @RT(0)
@END_Attrib
1 8 @F @F @F @F

@Var @RT(16)sv_LintabOutFwdV @RT(0) @T @T @DERIVED 0 @T @T @DT @RT(16)KAPPL_LintabData @RT(0) @T @T @UNKNOWN 0 @F
@F @F
@T
@BEG_Attrib
3 @RT(0) @RT(0) @RT(0)
@END_Attrib
1 8 @F @F @F @F

@Var @RT(16)sv_LintabOutBwdP @RT(0) @T @T @DERIVED 0 @T @T @DT @RT(16)KAPPL_LintabData @RT(0) @T @T @UNKNOWN 0 @F
@F @F
@T
@BEG_Attrib
3 @RT(0) @RT(0) @RT(0)
@END_Attrib
1 8 @F @F @F @F

@Var @RT(16)sv_LintabOutBwdV @RT(0) @T @T @DERIVED 0 @T @T @DT @RT(16)KAPPL_LintabData @RT(0) @T @T @UNKNOWN 0 @F
@F @F
@T
@BEG_Attrib
3 @RT(0) @RT(0) @RT(0)
@END_Attrib
1 8 @F @F @F @F

@Var @RT(15)sv_rMaxSpeedFwd @RT(0) @T @F @DT @RT(4)REAL @RT(0) @T @T @BASIC 0 @F
@F @F
@T
@BEG_Attrib
3 @RT(0) @RT(0) @RT(0)
@END_Attrib
1 8 @F @F @F @F

@Var @RT(15)sv_rMaxSpeedBwd @RT(0) @T @F @DT @RT(4)REAL @RT(0) @T @T @BASIC 0 @F
@F @F
@T
@BEG_Attrib
3 @RT(0) @RT(0) @RT(0)
@END_Attrib
1 8 @F @F @F @F

@Var @RT(15)sv_CylinderData @RT(0) @T @T @DERIVED 0 @T @T @DT @RT(14)tsCylinderData @RT(0) @T @T @UNKNOWN 0 @F
@F @F
@T
@BEG_Attrib
3 @RT(0) @RT(0) @RT(0)
@END_Attrib
1 8 @F @F @F @F

@Var @RT(18)sv_rMaxPressureFwd @RT(0) @T @F @DT @RT(4)REAL @RT(0) @T @T @BASIC 0 @F
@F @F
@T
@BEG_Attrib
3 @RT(0) @RT(0) @RT(0)
@END_Attrib
1 8 @F @F @F @F

@Var @RT(18)sv_rMaxPressureBwd @RT(0) @T @F @DT @RT(4)REAL @RT(0) @T @T @BASIC 0 @F
@F @F
@T
@BEG_Attrib
3 @RT(0) @RT(0) @RT(0)
@END_Attrib
1 8 @F @F @F @F

@Var @RT(19)sv_rMaxSpeedFwdCalc @RT(0) @T @T @RENAMED 0 @T @T @DT @RT(4)REAL @RT(0) @T @T @BASIC 0 @F
@F @F
@T
@BEG_Attrib
3 @RT(0) @RT(0) @RT(0)
@END_Attrib
1 8 @F @F @F @F

@Var @RT(19)sv_rMaxSpeedBwdCalc @RT(0) @T @T @RENAMED 0 @T @T @DT @RT(4)REAL @RT(0) @T @T @BASIC 0 @F
@F @F
@T
@BEG_Attrib
3 @RT(0) @RT(0) @RT(0)
@END_Attrib
1 8 @F @F @F @F

@Var @RT(20)sv_rMaxSpeedFwdCalib @RT(0) @T @T @RENAMED 0 @T @T @DT @RT(4)REAL @RT(0) @T @T @BASIC 0 @F
@F @F
@T
@BEG_Attrib
3 @RT(0) @RT(0) @RT(0)
@END_Attrib
1 8 @F @F @F @F

@Var @RT(20)sv_rMaxSpeedBwdCalib @RT(0) @T @T @RENAMED 0 @T @T @DT @RT(4)REAL @RT(0) @T @T @BASIC 0 @F
@F @F
@T
@BEG_Attrib
3 @RT(0) @RT(0) @RT(0)
@END_Attrib
1 8 @F @F @F @F

@Var @RT(25)sv_rMaxSpeedReducePercent @RT(0) @T @F @DT @RT(4)REAL @RT(0) @T @T @BASIC 0 @F
@F @F
@T
@BEG_Attrib
3 @RT(0) @RT(0) @RT(0)
@END_Attrib
1 8 @F @F @F @F

@Var @RT(15)miDigitsToFloor @RT(0) @T @F @DT @RT(4)SINT @RT(0) @T @T @BASIC 0 @F
@F @F
@T
@BEG_Attrib
3 @RT(1)2 @RT(0) @RT(0)
@END_Attrib
1 0 @F @F @F @F

@Var @RT(9)sv_bFALSE @RT(0) @T @F @DT @RT(4)BOOL @RT(0) @T @T @BASIC 0 @F
@F @F
@T
@BEG_Attrib
3 @RT(0) @RT(0) @RT(0)
@END_Attrib
1 8 @F @F @F @F

@END_Dcl

@END_Export

@BEG_Body

5

@BEG_Export

@BEG_Algo
@POSTUPDATE_ALGORITHM @RT(10)pInitStart @STRUCTURED_TEXT
@RT(0) @RT(13)sv_bInitStart @RT(9)PU_Task_7 @F @F
@END_Algo

@BEG_Dcl
@RT(16)DclTreeContainer
2
@Var @RT(18)abCalcMaxValuesFwd @RT(0) @T @T @DERIVED 0 @T @T @DT @RT(19)ABCalcHydrMaxValues @RT(0) @T @T @UNKNOWN 0 @F
@F @F
@T
@BEG_Attrib
3 @RT(0) @RT(0) @RT(0)
@END_Attrib
1 0 @F @F @F @F

@Var @RT(18)abCalcMaxValuesBwd @RT(0) @T @T @DERIVED 0 @T @T @DT @RT(19)ABCalcHydrMaxValues @RT(0) @T @T @UNKNOWN 0 @F
@F @F
@T
@BEG_Attrib
3 @RT(0) @RT(0) @RT(0)
@END_Attrib
1 0 @F @F @F @F

@END_Dcl

@END_Export

@BEG_Export

@BEG_Algo
@POSTUPDATE_ALGORITHM @RT(12)pDeviceStart @STRUCTURED_TEXT
@RT(0) @RT(15)sv_bDeviceStart @RT(9)EV_Task_1 @F @F
@END_Algo

@BEG_Dcl
@RT(16)DclTreeContainer
0
@END_Dcl

@END_Export

@BEG_Export

@BEG_Algo
@POSTUPDATE_ALGORITHM @RT(21)pInitRelLintabUpdater @STRUCTURED_TEXT
@RT(0) @RT(12)sv_bInitDone @RT(9)PU_Task_7 @F @F
@END_Algo

@BEG_Dcl
@RT(16)DclTreeContainer
4
@Var @RT(23)abUpdateRelLintabPreFwd @RT(0) @T @T @DERIVED 0 @T @T @DT @RT(20)ABUpdateRelLintabPre @RT(0) @T @T @UNKNOWN 0 @F
@F @F
@T
@BEG_Attrib
3 @RT(0) @RT(0) @RT(0)
@END_Attrib
1 0 @F @F @F @F

@Var @RT(23)abUpdateRelLintabVelFwd @RT(0) @T @T @DERIVED 0 @T @T @DT @RT(20)ABUpdateRelLintabVel @RT(0) @T @T @UNKNOWN 0 @F
@F @F
@T
@BEG_Attrib
3 @RT(0) @RT(0) @RT(0)
@END_Attrib
1 0 @F @F @F @F

@Var @RT(23)abUpdateRelLintabPreBwd @RT(0) @T @T @DERIVED 0 @T @T @DT @RT(20)ABUpdateRelLintabPre @RT(0) @T @T @UNKNOWN 0 @F
@F @F
@T
@BEG_Attrib
3 @RT(0) @RT(0) @RT(0)
@END_Attrib
1 0 @F @F @F @F

@Var @RT(23)abUpdateRelLintabVelBwd @RT(0) @T @T @DERIVED 0 @T @T @DT @RT(20)ABUpdateRelLintabVel @RT(0) @T @T @UNKNOWN 0 @F
@F @F
@T
@BEG_Attrib
3 @RT(0) @RT(0) @RT(0)
@END_Attrib
1 0 @F @F @F @F

@END_Dcl

@END_Export

@BEG_Export

@BEG_Algo
@PROCESS_ALGORITHM @RT(5)paRun @SEQUENTIAL_FLOW_CHART
@RT(0) @RT(0) @RT(16)TaskAnalog(5000) @F @F
@END_Algo

@BEG_Dcl
@RT(16)DclTreeContainer
2
@Var @RT(11)dActFwdTime @RT(0) @T @F @DT @RT(4)TIME @RT(0) @T @T @BASIC 0 @F
@F @F
@T
@BEG_Attrib
3 @RT(0) @RT(0) @RT(0)
@END_Attrib
1 4 @F @F @F @F

@Var @RT(1)b @RT(0) @T @F @DT @RT(4)BOOL @RT(0) @T @T @BASIC 0 @F
@F @F
@T
@BEG_Attrib
3 @RT(0) @RT(0) @RT(0)
@END_Attrib
1 4 @F @F @F @F

@END_Dcl

@END_Export

@BEG_Export

@BEG_Algo
@POSTUPDATE_ALGORITHM @RT(19)pActiveProfileStage @STRUCTURED_TEXT
@RT(0) @RT(31)sv_iActiveStage,sv_bDeviceReady @RT(9)PU_Task_3 @F @F
@END_Algo

@BEG_Dcl
@RT(16)DclTreeContainer
0
@END_Dcl

@END_Export

@BEG_Body
@TL(33)
(**************************************** WARNING ********************************************
 *** The KEBA Kemro K2 System including software is not intended for safety control tasks! ***
 ***                       For further information see Comment tab!                        ***
 *********************************************************************************************)

IF sv_bInitStart THEN

   //check if transducer is available
   sv_bTransducerAvailable := IS_LINKED(ai_Position);
   IF (sv_bTransducerAvailable) THEN
      sv_Options := sv_Options OR cSubOpNozzleTransducer;
      //set auto-calib transducer
      sv_CalibState.prInputSensor := @ai_Position;
   END_IF;

   //register and init nozzle bwd movement
   abMoveBwd.aRegister();
   abMoveBwd.aInit();

   //register and init nozzle fwd movement
   abMoveFwd.aRegister();
   abMoveFwd.aInit();

   //init calculation of hydraulic max values for nozzle fwd
   abCalcMaxValuesFwd.aInit(pRequiredPumps := @sv_RequiredPumpsFwd,
                            pHydrMaxValues := @sv_HydrMaxValuesFwd);

   //init calculation of hydraulic max values for nozzle bwd
   abCalcMaxValuesBwd.aInit(pRequiredPumps := @sv_RequiredPumpsBwd,
                            pHydrMaxValues := @sv_HydrMaxValuesBwd);

END_IF;

@END_Body

@@@BEG_Comment@@@
@TL(2)
Calls the registration-algo of every movementblock after the deviceregistration succeeded(sv_bInitStart->true)

@@@END_Comment@@@

@BEG_Body
@TL(10)
(**************************************** WARNING ********************************************
 *** The KEBA Kemro K2 System including software is not intended for safety control tasks! ***
 ***                       For further information see Comment tab!                        ***
 *********************************************************************************************)

IF sv_bDeviceStart THEN
   //start device
   START_PROCESS_ALGORITHM(paRun);
END_IF;

@END_Body

@@@BEG_Comment@@@
@TL(1)
Starts the algo paRun when sv_bDeviceStart is set by ABControl.
@@@END_Comment@@@

@BEG_Body
@TL(39)
(**************************************** WARNING ********************************************
 *** The KEBA Kemro K2 System including software is not intended for safety control tasks! ***
 ***                       For further information see Comment tab!                        ***
 *********************************************************************************************)

abUpdateRelLintabPreFwd.aInit(pLintabOut := @sv_LintabOutFwdP,
                              prMaxPressure := @sv_rMaxPressureFwd,
                              prMaxHydrPressure := @sv_HydrMaxValuesFwd.rMaxPressure,
                              bUseForce := TRUE,
                              bFwd := TRUE,
                              pCylinderData := @sv_CylinderData);

abUpdateRelLintabVelFwd.aInit(pLintabOut := @sv_LintabOutFwdV,
                              prMaxSpeed := @sv_rMaxSpeedFwd,
                              prMaxSpeedCalc := @sv_rMaxSpeedFwdCalc,
                              prMaxSpeedCalib := @sv_rMaxSpeedFwdCalib,
                              prMaxSpeedReducePercent := @sv_rMaxSpeedReducePercent,
                              iMaxSpeedDigitsToFloor := miDigitsToFloor,
                              prAbsFlow := @sv_HydrMaxValuesFwd.rAbsFlow,
                              bFwd := TRUE,
                              pCylinderData := @sv_CylinderData);

abUpdateRelLintabPreBwd.aInit(pLintabOut := @sv_LintabOutBwdP,
                              prMaxPressure := @sv_rMaxPressureBwd,
                              prMaxHydrPressure := @sv_HydrMaxValuesBwd.rMaxPressure,
                              bUseForce := TRUE,
                              bFwd := FALSE,
                              pCylinderData := @sv_CylinderData);

abUpdateRelLintabVelBwd.aInit(pLintabOut := @sv_LintabOutBwdV,
                              prMaxSpeed := @sv_rMaxSpeedBwd,
                              prMaxSpeedCalc := @sv_rMaxSpeedBwdCalc,
                              prMaxSpeedCalib := @sv_rMaxSpeedBwdCalib,
                              prMaxSpeedReducePercent := @sv_rMaxSpeedReducePercent,
                              iMaxSpeedDigitsToFloor := miDigitsToFloor,
                              prAbsFlow := @sv_HydrMaxValuesBwd.rAbsFlow,
                              bFwd := FALSE,
                              pCylinderData := @sv_CylinderData);

@END_Body

@@@BEG_Comment@@@
@TL(0)

@@@END_Comment@@@

@BEG_SfcBody
19 18 21

@BEG_SfcData 2
@StepSeq @RT(4)sseq @F 1
@Loop @RT(4)loop @F 2
@StepSeq @RT(3)seq @F 5
@Step @RT(5)START @F @T @F @F @RT(0) @F
@AcbCont @RT(7)unnamed @F 1
@Acb @RT(8)Action18 @F @T @RT(1)P @RT(0) @F @F @T @TL(2)
b := WRITE_SV_DIRECT(sv_bDeviceStart, sv_bFALSE);

@F

@Trans @RT(6)TStart @F @T @F @F @T @F @TL(2)
TRUE

@RT(7)Trans12 @F
@Step @RT(14)OUTPUT_REQUEST @F @F @F @F @RT(0) @F
@AcbCont @RT(7)unnamed @F 2
@Acb @RT(14)AOutputRequest @F @T @RT(1)P @RT(0) @F @F @T @TL(3)
abOutputRequest.aRequest(pMoveData := g_MoveCtrl.pData,
                         AnaOutputMode := nAnaOutputModeMid);

@F
@Acb @RT(12)ACheckOutput @F @T @RT(1)N @RT(0) @F @F @T @TL(2)
abOutputRequest.aCheck();

@F

@AltBranch @RT(3)alt @F 2
@TransSeq @RT(4)tseq @F 1
@Trans @RT(7)Trans13 @F @T @F @F @T @T @TL(2)
g_MoveCtrl.bStop

@RT(7)Trans13 @F

@TransSeq @RT(4)tseq @F 3
@Trans @RT(7)Trans15 @F @T @F @F @T @F @TL(2)
abOutputRequest.aCheck.bReady

@RT(7)Trans15 @F
@Step @RT(6)OUTPUT @F @F @F @F @RT(0) @F
@AcbCont @RT(7)unnamed @F 0

@AltBranch @RT(3)alt @F 2
@TransSeq @RT(4)tseq @F 3
@Trans @RT(6)Trans9 @F @T @F @F @T @F @TL(2)
g_MoveCtrl.pData^.MoveDir = cMoveBwd

@RT(6)Trans9 @F
@Step @RT(3)BWD @F @F @F @F @RT(0) @F
@AcbCont @RT(7)unnamed @F 1
@Acb @RT(4)aBwd @F @F @RT(1)N @RT(0) @F @F @T @F

@Trans @RT(9)TBwdReady @F @T @F @F @T @F @TL(2)
abMoveBwd.aRun.bReady;

@RT(6)Trans1 @F

@TransSeq @RT(4)tseq @F 3
@Trans @RT(6)Trans2 @F @T @F @F @T @F @TL(2)
g_MoveCtrl.pData^.MoveDir = cMoveFwd

@RT(6)Trans2 @F
@Step @RT(3)FWD @F @F @F @F @RT(0) @F
@AcbCont @RT(7)unnamed @F 1
@Acb @RT(4)aFwd @F @F @RT(1)N @RT(0) @F @F @T @F

@Trans @RT(9)TFwdReady @F @T @F @F @T @F @TL(2)
abMoveFwd.aRun.bReady

@RT(7)Trans11 @F

@Step @RT(5)READY @F @F @F @F @RT(0) @F
@AcbCont @RT(7)unnamed @F 1
@Acb @RT(7)Action2 @F @T @RT(1)P @RT(0) @F @F @T @TL(6)
abOutputRequest.aRelease(pMoveData := g_MoveCtrl.pData);
g_MoveCtrl.bReady := TRUE;
IF NOT sv_bDeviceStart THEN
    STOP_PROCESS_ALGORITHM();
END_IF;

@F

@Trans @RT(6)Trans8 @F @T @T @T @T @T @TL(2)
TRUE

@RT(6)Trans8 @F

@END_SfcData
@SaActions 2
@SaText @RT(4)aBwd 1 @TL(7)
(**************************************** WARNING ********************************************
 *** The KEBA Kemro K2 System including software is not intended for safety control tasks! ***
 ***                       For further information see Comment tab!                        ***
 *********************************************************************************************)

abMoveBwd.aRun(bStop := g_MoveCtrl.bStop);

@SaText @RT(4)aFwd 1 @TL(7)
abMoveFwd.aRun(bStop := g_MoveCtrl.bStop);

IF g_MoveCtrl.pData^.MoveId = cMoveFwdContactF THEN
   dActFwdTime := FWD.T;
   b := WRITE_SV_DIRECT(sv_dActFwdTime, dActFwdTime);
END_IF;

@SaTrans 0
@SaExits 0
@END_SfcBody

@@@BEG_Comment@@@
@TL(3)
Calls depending on the MoveId and MoveDir the movementblock. g_MoveCtrl.MoveId/MoveDir are set by the Block ABControl after
evStart was received. The movement-block has to be called until the it returns abMoveXxx.aRun.bReady.
In case of hydraulic movements the output-request has to be done before starting the movement.
@@@END_Comment@@@

@BEG_Body
@TL(40)
(**************************************** WARNING ********************************************
 *** The KEBA Kemro K2 System including software is not intended for safety control tasks! ***
 ***                       For further information see Comment tab!                        ***
 *********************************************************************************************)

IF NOT sv_bDeviceReady THEN

   IF sv_OperationMode = nSetup THEN
      //movement in setup mode active
      //-> reset active stage information
      sv_iActiveStageFwd := 0;
      sv_iActiveStageBwd := 0;
   ELSE

      //nozzle movement in manual - half - or fullauto mode
      IF g_MoveCtrl.pData^.MoveDir = cMoveFwd THEN

         //reset bwd stage info if fwd movement is started
         sv_iActiveStageBwd := 0;

         IF sv_iActiveStage > 0 THEN
            sv_iActiveStageFwd := sv_iActiveStage;
         END_IF;

      ELSIF g_MoveCtrl.pData^.MoveDir = cMoveBwd THEN

         //reset Fwd stage info if bwd movement is started
         sv_iActiveStageFwd := 0;

         IF sv_iActiveStage > 0 THEN
            sv_iActiveStageBwd := sv_iActiveStage;
         END_IF;
      END_IF;
   END_IF;

END_IF;

@END_Body

@@@BEG_Comment@@@
@TL(0)

@@@END_Comment@@@
@END_Body

@END_Contents
